// TIA Portal project "OPC_try" (V15.1)

(* hardware
DEVICE "S71500/ET200MP station_1"  S7-1500 station
   slot 0: "Rail_0"  Rack  6ES7 590-1***0-0AA0
   slot 1: "PLC_1"  CPU 1516-3 PN/DP  6ES7 516-3AN01-0AB0  V2.6
      slot 3: "CPU display_1"  6ES7591-1BA00-0AA0
   slot 2: "AI 8xU/I/RTD/TC ST_1"  AI 8xU/I/RTD/TC ST  6ES7 531-7KF00-0AB0  V2.2
   slot 3: "AQ 4xU/I ST_1"  AQ 4xU/I ST  6ES7 532-5HD00-0AB0  V2.2
   slot 4: "DI 32x24VDC HF_1"  DI 32x24VDC HF  6ES7 521-1BL00-0AB0  V2.1
   slot 5: "DQ 32x24VDC/0.5A HF_1"  DQ 32x24VDC/0.5A HF  6ES7 522-1BL01-0AB0  V1.1
*)

// ===== PLC "PLC_1"  CPU 1516-3 PN/DP =====

VAR_GLOBAL   // PLC tag table "Default tag table"
   "Tag_1" AT %Q19.7 : Bool;
   "Tag_2" AT %Q9.7 : Bool;
   "Tag_3" AT %I17.4 : Bool;
END_VAR

DATA_BLOCK "Prueba_OPC"   // DB1
{ S7_Optimized_Access := 'TRUE' }
VERSION : 0.1
   VAR
      Prueba_OPC_INT : Int;
      Prueba_OPC_BOOL : Bool;
   END_VAR
BEGIN
END_DATA_BLOCK

ORGANIZATION_BLOCK "Main"   // OB1, LAD, ProgramCycle
TITLE = "Main Program Sweep (Cycle)"
{ S7_Optimized_Access := 'TRUE' }
VERSION : 0.1
   VAR_INPUT
      Initial_Call : Bool;   // Initial call of this OB
      Remanence : Bool;   // =True, if remanent data are available
   END_VAR
BEGIN

REGION Network 1
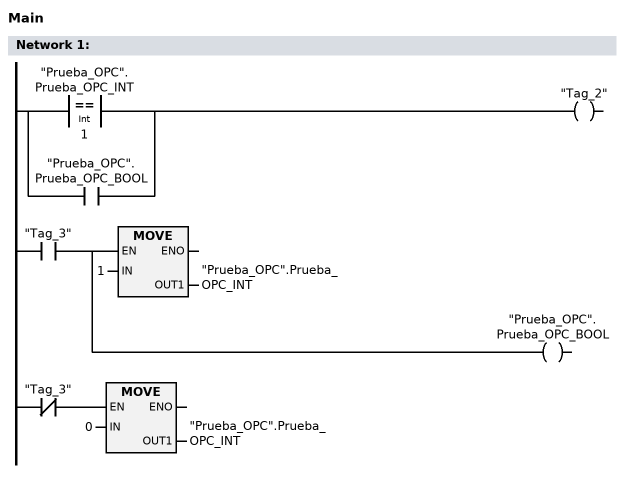
   RUNG wire#powerrail
      { S7_Templates := "SrcType := Int" } EQ_Contact(in1 := "Prueba_OPC".Prueba_OPC_INT, in2 := 1)
      wire#w1
      Coil( "Tag_2" )
   END_RUNG
   RUNG wire#powerrail
      Contact( "Prueba_OPC".Prueba_OPC_BOOL )
   END_RUNG wire#w1
   RUNG wire#powerrail
      Contact( "Tag_3" )
      wire#w2
      Move(in := 1, out1 => "Prueba_OPC".Prueba_OPC_INT)
   END_RUNG
   RUNG wire#w2
      Coil( "Prueba_OPC".Prueba_OPC_BOOL )
   END_RUNG
   RUNG wire#powerrail
      I_Contact( "Tag_3" )
      Move(in := 0, out1 => "Prueba_OPC".Prueba_OPC_INT)
   END_RUNG
   // the same network as SCL:
   "Tag_2" := ("Prueba_OPC".Prueba_OPC_INT = 1) OR "Prueba_OPC".Prueba_OPC_BOOL;
   IF "Tag_3" THEN "Prueba_OPC".Prueba_OPC_INT := 1; END_IF;
   "Prueba_OPC".Prueba_OPC_BOOL := "Tag_3";
   IF NOT "Tag_3" THEN "Prueba_OPC".Prueba_OPC_INT := 0; END_IF;
END_REGION
END_ORGANIZATION_BLOCK